PROGRAM A01_StartupBridge
VAR
	fbStartBridge: NT_StartProcess;
	fbPulse: FB_SquareWave;
	tonNotRunning: TON;
	bBusyOnce	:BOOL;

	ton_Watchdog: TON;
	nLastWatchdogFromBridge	: DINT;
	bWait: BOOL;

	bBridgeLocalRun : BOOL;

END_VAR


(*
Modification history:
Date		|	Author 		|	Remark
----------------------------------------------------------------------------------------------------
03.09.20	|	PP			|	Start Remarking.
*)

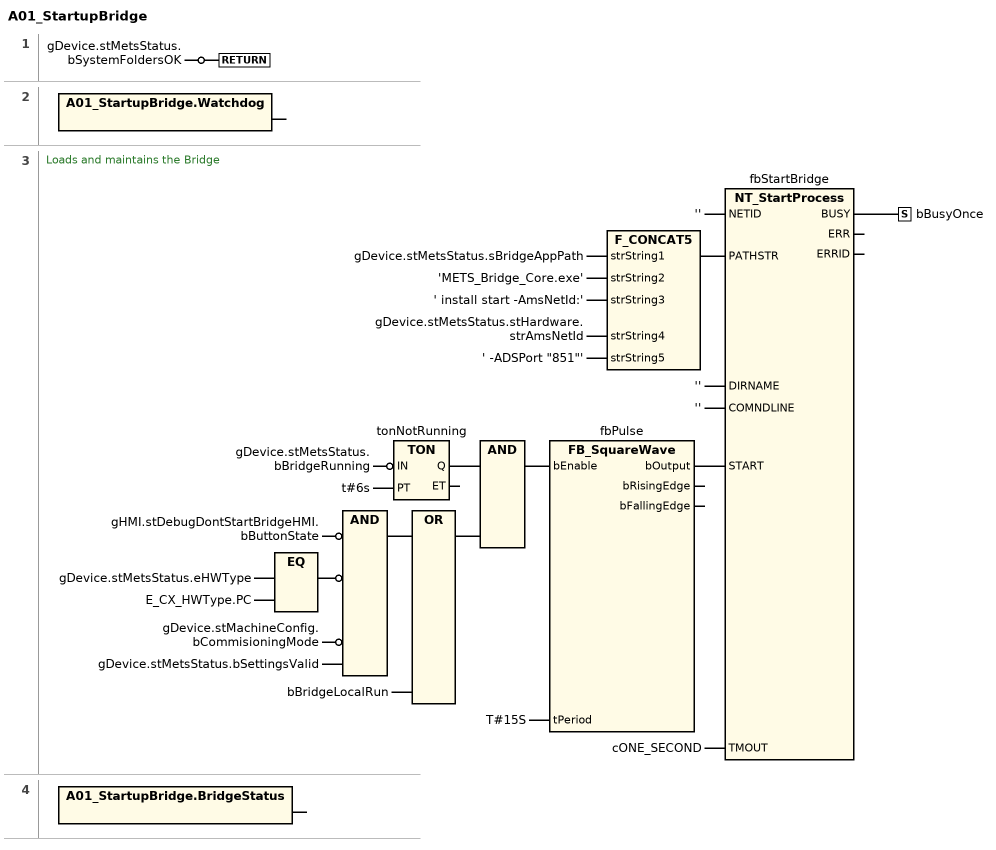
// NETWORK 1
IF NOT gDevice.stMetsStatus.bSystemFoldersOK THEN RETURN; END_IF

// NETWORK 2
A01_StartupBridge.Watchdog();

// NETWORK 3
// Loads and maintains the Bridge
tonNotRunning(IN := NOT gDevice.stMetsStatus.bBridgeRunning, PT := t#6s); // TON
fbPulse(bEnable := tonNotRunning.Q AND (NOT gHMI.stDebugDontStartBridgeHMI.bButtonState AND NOT (gDevice.stMetsStatus.eHWType = E_CX_HWType.PC) AND NOT gDevice.stMachineConfig.bCommisioningMode AND gDevice.stMetsStatus.bSettingsValid OR bBridgeLocalRun), tPeriod := T#15S); // FB_SquareWave
fbStartBridge(
    NETID := '',
    PATHSTR := F_CONCAT5(strString1 := gDevice.stMetsStatus.sBridgeAppPath, strString2 := 'METS_Bridge_Core.exe', strString3 := ' install start -AmsNetId:', strString4 := gDevice.stMetsStatus.stHardware.strAmsNetId, strString5 := ' -ADSPort "851"'),
    DIRNAME := '',
    COMNDLINE := '',
    START := fbPulse.bOutput,
    TMOUT := cONE_SECOND); // NT_StartProcess
bBusyOnce S= fbStartBridge.BUSY;

// NETWORK 4
A01_StartupBridge.BridgeStatus();

ACTION BridgeStatus:
//{warning 'CONVERSION MESSAGE: This text contained unprintable characters, that have been deleted'.}
(* nBridgeStatus:
Initialized = 0, 
TwincatInitialized = 1, 
PLCVariablesInitialized = 2, 
ReadProcessVariablesError = 3, 
PCMReceiverInitialized = 4,  
PCMReceiverRunning = 5, 
PCMReceiverNewPCMArrived = 6, 
ServiceError = 7, 
BridgeInCommissioningMode = 8, 
BridgeConnectedToFSS = 9*)

gDevice.stMetsStatus.bPCMReceiverRunning	:= gDevice.stBridge.nBridgeStatus.5;
gDevice.stMetsStatus.bMETSConnectedToFSS 	:= gDevice.stBridge.nBridgeStatus.9;

gPersistent.sLastFileNameToDlogHMI			:= gDevice.stBridge.sLastFileNameToDlogHMI;
gPersistent.sLastFileTimeToDlogHMI			:= gDevice.stBridge.sLastFileTimeToDlogHMI;

gDevice.stBridge.sFSSServerIpAddress 		:= gDevice.stMachineConfig.sFSS_Server_IPAddress;
gDevice.stBridge.sFSSServerWebRequest 		:= gDevice.stMachineConfig.sFSS_Server_WebRequest;

gDevice.stBridge.nFSSResponseTimeout 		:= gDevice.stMachineConfig.nFSSResponseTimeout;
gDevice.stBridge.nFSSResendAttempts 		:= gDevice.stMachineConfig.nFSSResendAttempts;
gDevice.stBridge.bCommissioningMode 		:= gDevice.stMachineConfig.bCommisioningMode;

gDevice.stBridge.sFaultCodeDirectory 		:= gDevice.stMetsStatus.sMETSProcessPath;
gDevice.stBridge.sFSSFaultCodeAge 			:= 10;
gDevice.stBridge.sFSSCHMDirectory 			:= gDevice.stMetsStatus.sCHMPath;
gDevice.stBridge.nBridgeTimeout				:= 1000;

(*gDevice.stBridge.sDBConnectionString			:= stDBStatus.sDBConnectionString;*)
gDevice.stBridge.sLocalCACPath				:= gDevice.stMetsStatus.sCACPath;
gDevice.stBridge.sLocalBridgePath			:= gDevice.stMetsStatus.sBridgeAppPath;
END_ACTION

ACTION Watchdog:
(*Watchdog to Bridge*)
gDevice.nWatchdogToBridge := gDevice.nWatchdogToBridge + 1;
IF  gDevice.nWatchdogToBridge > 100000 THEN
	gDevice.nWatchdogToBridge := 1;
END_IF

gDevice.nWatchdogFromBridge	:=	gDevice.stBridge.nBridgeWatchdog;
(*Watchdog from HMI - check if running*)
IF ton_Watchdog.Q THEN
	bWait := FALSE;
	IF gDevice.nWatchdogFromBridge <> nLastWatchdogFromBridge THEN
		gDevice.stMetsStatus.bBridgeRunning := TRUE;
		nLastWatchdogFromBridge := gDevice.nWatchdogFromBridge;
	ELSE
		gDevice.stMetsStatus.bBridgeRunning := FALSE;
	END_IF
ELSE
	bWait := TRUE;
END_IF

ton_Watchdog(IN:= bWait, PT := t#4000ms);
END_ACTION

END_PROGRAM

(* stored: Version 1.1.0.1
   POU A01_StartupBridge: Id {64573b79-04f9-49c2-8bd2-a375674dd269}, SpecialFunc None
   Action BridgeStatus: Id {3ee8bfd6-f26c-45bb-ba5a-368c8b54597b}
   Action Watchdog: Id {7bf25c63-a202-4109-b87a-fca27f5f33ba} *)
